FUNCTION_BLOCK ManipulateFunctionsTest EXTENDS TcUnit.FB_TestSuite
VAR
END_VAR

ClearDataFunction();
ShiftDataLeftFunction();
ShiftDataRightFunction();
SwapFunction();
SwapByPointerFunction();

METHOD ClearDataFunction : BOOL
VAR
	data : INT;
END_VAR
TcUnit.TEST('Clear data function');

data := 42;
ClearData(data);

AssertEquals_INT(
	Expected := 0,
	Actual := data,
	Message := 'Data memory should be all set to 0');

TEST_FINISHED();
END_METHOD

METHOD ShiftDataLeftFunction : BOOL
VAR
	updatedBuffer : ARRAY[0..LastIndex] OF INT;
	
	expected : ARRAY[0..LastIndex] OF INT;
END_VAR
VAR CONSTANT
	LastIndex : INT := 2;
END_VAR
TcUnit.TEST('Shift data left function');

updatedBuffer[LastIndex] := 1;
ShiftDataLeft(updatedBuffer, SIZEOF(INT));
updatedBuffer[LastIndex] := 2;
ShiftDataLeft(updatedBuffer, SIZEOF(INT));
updatedBuffer[LastIndex] := 3;

expected[0] := 1;
expected[1] := 2;
expected[2] := 3;

AssertArrayEquals_INT(
	Expecteds := expected,
	Actuals := updatedBuffer,
	Message := 'Data should be gradually shifter from end to begin');

TEST_FINISHED();
END_METHOD

METHOD ShiftDataRightFunction : BOOL
VAR
	updatedBuffer : ARRAY[0..LastIndex] OF INT;
	
	expected : ARRAY[0..LastIndex] OF INT;
END_VAR
VAR CONSTANT
	LastIndex : INT := 2;
END_VAR
TcUnit.TEST('Shift data right function');

updatedBuffer[0] := 3;
ShiftDataRight(updatedBuffer, SIZEOF(INT));
updatedBuffer[0] := 2;
ShiftDataRight(updatedBuffer, SIZEOF(INT));
updatedBuffer[0] := 1;

expected[0] := 1;
expected[1] := 2;
expected[2] := 3;

AssertArrayEquals_INT(
	Expecteds := expected,
	Actuals := updatedBuffer,
	Message := 'Data should be gradually shifter from begin to end');

TEST_FINISHED();
END_METHOD

METHOD SwapByPointerFunction : BOOL
VAR
	data1 : INT;
	data2 : INT;
END_VAR
TcUnit.TEST('Swap by pointer function');

data1 := 42;
data2 := 420;

SwapByPointer(ADR(data1), ADR(data2), SIZEOF(data1));

AssertEquals_BOOL(
	Expected := TRUE,
	Actual := data1 = 420 AND data2 = 42,
	Message := 'Data should be swapped');

TEST_FINISHED();
END_METHOD

METHOD SwapFunction : BOOL
VAR
	data1 : INT;
	data2 : INT;
END_VAR
TcUnit.TEST('Swap function');

data1 := 42;
data2 := 420;

Swap(data1, data2);

AssertEquals_BOOL(
	Expected := TRUE,
	Actual := data1 = 420 AND data2 = 42,
	Message := 'Data should be swapped');

TEST_FINISHED();
END_METHOD

END_FUNCTION_BLOCK

(* stored: Version 1.1.0.1, ProductVersion 3.1.4024.15
   POU ManipulateFunctionsTest: Id {1f377edf-7d66-0e65-08df-d611dbb1e58f}, SpecialFunc None
   Method ClearDataFunction: Id {deb98a0e-9a2e-064c-13db-bf7d3fda682e}
   Method ShiftDataLeftFunction: Id {882b59ca-147e-020a-1cd6-c9e4161e4350}
   Method ShiftDataRightFunction: Id {c2ae2d3d-03c5-0645-2dda-2dd651203613}
   Method SwapByPointerFunction: Id {7193cf85-b820-060b-0903-250304d7c7f2}
   Method SwapFunction: Id {9bc59df5-58cc-0cb9-3186-8a72c385a324} *)
